//Größendimension von Objecten
TYPE ST_3DDimension :	
STRUCT
	Width  : REAL;	//Breite in µm
	Depth  : REAL;	//Tiefe in µm
	Height : REAL;	//Höhe in µm	
END_STRUCT
END_TYPE

(* stored: Version 1.1.0.1, ProductVersion 3.1.0.23
   DUT ST_3DDimension: Id {c3dc4f75-a58e-4063-a411-4f1d4fea963f} *)
